// TIA Portal project "FactoryIO_Template_S7-1200_V15_V15.1" (V15.1)
// Vorlageprojekt für das Buch mit Zielsystem S7-1200

(* hardware
DEVICE "S7-1200-Station_1"  S7-1200 Station
   slot 0: "Baugruppenträger_0"  Rack  V1.0
   slot 1: "PLC_1"  CPU 1211C DC/DC/DC  6ES7 211-1AE40-0XB0  V4.1
DEVICE "HMI_1"  KTP700 Basic PN
   slot 0: "HMI_1"  KTP700 Basic PN  6AV2 123-2GB03-0AX0  15.1.0.0
   slot 1: "HMI_RT_1"  KTP700 Basic PN  6AV2 123-2GB03-0AX0  15.1.0.0
   slot 5: "HMI_1.IE_CP_1"  PROFINET Interface  15.0.1.0
      slot 1: "Interfaz PROFINET_1"  PROFINET Interface
         slot 1: "Port_1"  Port
*)

// ===== PLC "PLC_1"  CPU 1211C DC/DC/DC =====

VAR_GLOBAL   // PLC tag table "Standard-Variablentabelle"
   "Start" AT %I0.3 : Bool;
   "Reset" AT %I0.4 : Bool;
   "Stop" AT %I0.5 : Bool;
   "Auto" AT %I0.6 : Bool;
   "Emergency Stop" AT %I0.7 : Bool;
   "Buffer vel" AT %ID30 : Real;
   "At buffer entry" AT %I0.0 : Bool;
   "At buffer exit" AT %I0.1 : Bool;
   "At exit" AT %I0.2 : Bool;
   "Stop Blade" AT %Q0.0 : Bool;
   "Start Light" AT %Q0.1 : Bool;
   "Reset Light" AT %Q0.2 : Bool;
   "Stop Light" AT %Q0.3 : Bool;
   "Emitter" AT %Q0.4 : Bool;
   "Buffer Conveyor" AT %QD30 : Real;
   "Exit Conveyor" AT %QD34 : Real;
   "Counter" AT %QD38 : DInt;
   "System_Byte" AT %MB1 : Byte;
   "FirstScan" AT %M1.0 : Bool;
   "DiagStatusUpdate" AT %M1.1 : Bool;
   "AlwaysTRUE" AT %M1.2 : Bool;
   "AlwaysFALSE" AT %M1.3 : Bool;
   "System_Byte(1)" AT %MB1 : Byte;
   "Clock_Byte" AT %MB0 : Byte;
   "Clock_10Hz" AT %M0.0 : Bool;
   "Clock_5Hz" AT %M0.1 : Bool;
   "Clock_2.5Hz" AT %M0.2 : Bool;
   "Clock_2Hz" AT %M0.3 : Bool;
   "Clock_1.25Hz" AT %M0.4 : Bool;
   "Clock_1Hz" AT %M0.5 : Bool;
   "Clock_0.625Hz" AT %M0.6 : Bool;
   "Clock_0.5Hz" AT %M0.7 : Bool;
   "Started State" AT %M2.0 : Bool;
   "Reset State" AT %M2.1 : Bool;
   "Stop State" AT %M2.2 : Bool;
   "Emergency Stop State" AT %M2.3 : Bool;
   "Emergency Rearm State" AT %M2.4 : Bool;
   "Norm input" AT %MD30 : Real;
   "Half vel" AT %MD34 : Real;
   "Counter Entry" AT %MD50 : DInt;
   "Counter Exit" AT %MD54 : DInt;
   "Transitioning State" AT %M3.0 : Bool;
   "Exiting State" AT %M3.1 : Bool;
   "Forzar Entrada" AT %M2.5 : Bool;
   "Forzar Valor" AT %MD38 : Real;
   "Start HMI" AT %M2.6 : Bool;
   "Stop HMI" AT %M2.7 : Bool;
   "Tag_1" AT %M3.2 : Bool;
   "Tag_2" AT %M3.3 : Bool;
   "Tag_3" AT %MD42 : Real;
   "Tag_4" AT %MD46 : Real;
   "Tag_5" AT %MD58 : Real;
   "Tag_6" AT %MD62 : Real;
   "Tag_7" AT %MD66 : Real;
   "Tag_8" AT %MD70 : Real;
END_VAR

// folder: System blocks/Program resources

DATA_BLOCK "IEC_Timer_0_DB"   // DB1
{ S7_Optimized_Access := 'TRUE' }
AUTHOR : Simatic
FAMILY : IEC
NAME : IEC_TMR
VERSION : 1.0
// stored: InstanceOfName IEC_TIMER
"IEC_TIMER"
BEGIN
END_DATA_BLOCK

DATA_BLOCK "IEC_Counter_0_DB"   // DB2
{ S7_Optimized_Access := 'TRUE' }
AUTHOR : SIMATIC
FAMILY : IEC
NAME : DCNTR
VERSION : 1.2
// stored: InstanceOfName IEC_DCOUNTER
"IEC_DCOUNTER"
BEGIN
END_DATA_BLOCK

DATA_BLOCK "IEC_Counter_0_DB_1"   // DB3
{ S7_Optimized_Access := 'TRUE' }
AUTHOR : SIMATIC
FAMILY : IEC
NAME : DCNTR
VERSION : 1.2
// stored: InstanceOfName IEC_DCOUNTER
"IEC_DCOUNTER"
BEGIN
END_DATA_BLOCK

// folder: (top level)

FUNCTION "MHJ-PLC-Lab-Function-S71200" : Void   // FC9000, SCL
{ S7_Optimized_Access := 'TRUE' }
VERSION : 0.1
   VAR_TEMP
      rdTimeReturn : Int;
      outputTime : DTL;
      SyncVal : Byte;
      forVal : Int;
      forVal_2 : Int;
      Value : Byte;
   END_VAR
   VAR CONSTANT
      CompVal : Byte := 16#34;
      Value_01 : Byte := 16#11;
      Value_01_DW : DWord := 16#A165_D992;
      Value_02_DW : DWord := 16#58BE_4401;
   END_VAR
BEGIN

   #Value:=PEEK(area := 16#82,
        dbNumber := 0,
        byteOffset := 511);
   #Value := #Value + 1;

   POKE(area := 16#82,
        dbNumber := 0,
        byteOffset := 511,
        value := #Value);

   POKE(area:=16#81,
        dbNumber:=0,
        byteOffset:=1016,
        value:=#Value_01_DW);
   POKE(area := 16#81,
        dbNumber := 0,
        byteOffset := 1020,
        value := #Value_02_DW);

   POKE(area := 16#81,
        dbNumber := 0,
        byteOffset := 511,
        value := B#16#00);

   FOR #forVal := 0 TO 120 DO
       FOR #forVal_2:=0 TO 10 DO
           #rdTimeReturn:=RD_SYS_T(#outputTime);
           #rdTimeReturn := WR_SYS_T(#outputTime);
           #rdTimeReturn := RD_SYS_T(#outputTime);
           #rdTimeReturn := WR_SYS_T(#outputTime);
       END_FOR;
       #SyncVal:= PEEK(area := 16#81,
                      dbNumber := 0,
                      byteOffset := 511);
       IF #SyncVal = #CompVal THEN
          GOTO M_1;
       END_IF;
   END_FOR;
   RETURN;

   M_1:
   POKE(area := 16#81,
        dbNumber := 0,
        byteOffset := 511,
        value := B#16#0);
END_FUNCTION

ORGANIZATION_BLOCK "Main"   // OB1, LAD, ProgramCycle
TITLE = "Main Program Sweep (Cycle)"
{ S7_Optimized_Access := 'TRUE' }
VERSION : 0.1
   VAR_INPUT
      Initial_Call : Bool;   // Initial call of this OB
      Remanence : Bool;   // =True, if remanent data are available
   END_VAR
   VAR_TEMP   // added for the SCL form of the ladder/FBD networks
      _w1 : Bool;
      _w2 : Bool;
      _w3 : Bool;
      _w4 : Bool;
      _w5 : Bool;
      _w6 : Bool;
      _w7 : Bool;
      _w8 : Bool;
   END_VAR
BEGIN

REGION Network 1: Konnektierungsbaustein für PLC-Lab / Comunicacion con Factory IO (no tocar)
   // Im Netzwerk 1 wird der Konnektierungsbaustein für PLC-Lab aufgerufen.
   // Dieser Aufruf darf nicht entfernt werden!
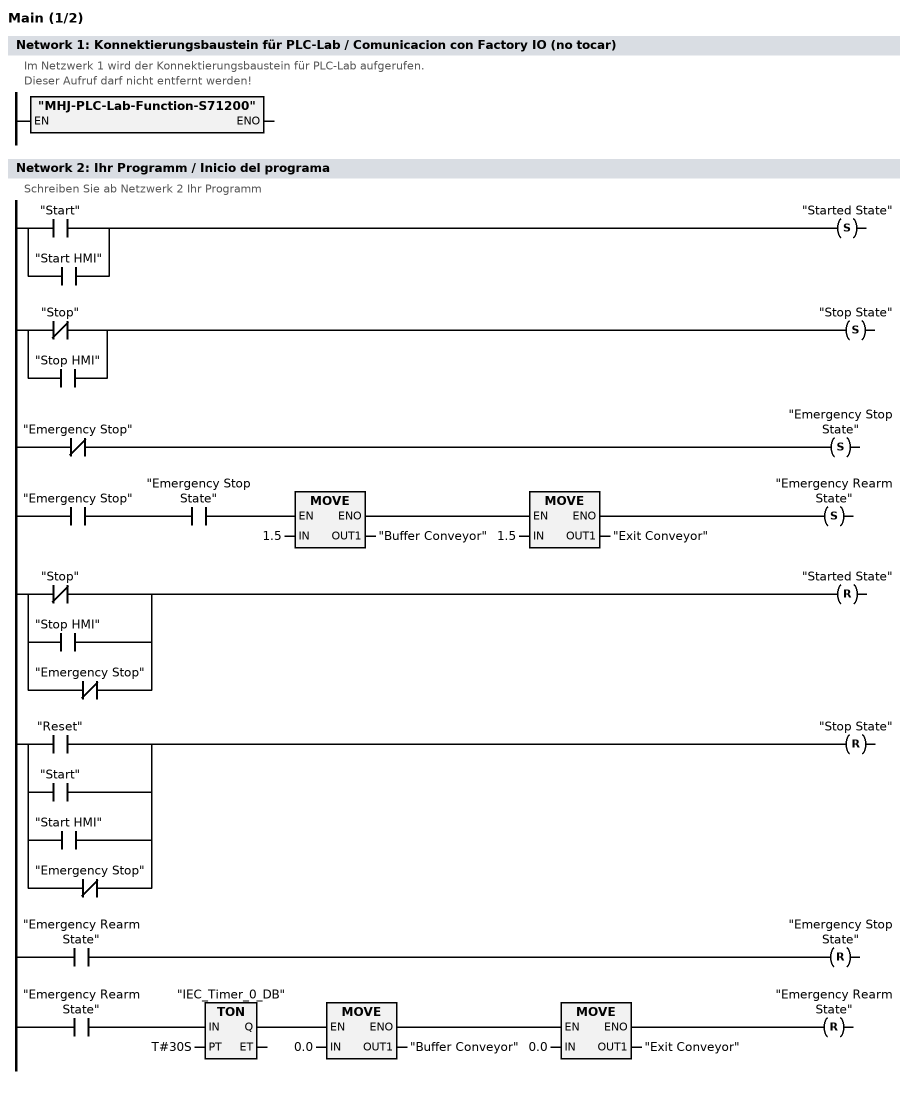
   RUNG wire#powerrail
      "MHJ-PLC-Lab-Function-S71200"()
   END_RUNG
   // the same network as SCL:
   "MHJ-PLC-Lab-Function-S71200"();
END_REGION

REGION Network 2: Ihr Programm / Inicio del programa
   // Schreiben Sie ab Netzwerk 2 Ihr Programm
   IF "Start" OR "Start HMI" THEN "Started State" := TRUE; END_IF;
   IF NOT "Stop" OR "Stop HMI" THEN "Stop State" := TRUE; END_IF;
   IF NOT "Emergency Stop" THEN "Emergency Stop State" := TRUE; END_IF;
   IF "Emergency Stop" AND "Emergency Stop State" THEN
       "Buffer Conveyor" := 1.5;
       "Exit Conveyor" := 1.5;
       "Emergency Rearm State" := TRUE;
   END_IF;
   IF NOT "Stop" OR "Stop HMI" OR NOT "Emergency Stop" THEN "Started State" := FALSE; END_IF;
   IF "Reset" OR "Start" OR "Start HMI" OR NOT "Emergency Stop" THEN "Stop State" := FALSE; END_IF;
   IF "Emergency Rearm State" THEN "Emergency Stop State" := FALSE; END_IF;
   "IEC_Timer_0_DB".TON(IN := "Emergency Rearm State", PT := T#30S);
   IF "IEC_Timer_0_DB".Q THEN
       "Buffer Conveyor" := 0.0;
       "Exit Conveyor" := 0.0;
       "Emergency Rearm State" := FALSE;
   END_IF;
END_REGION

REGION Network 3
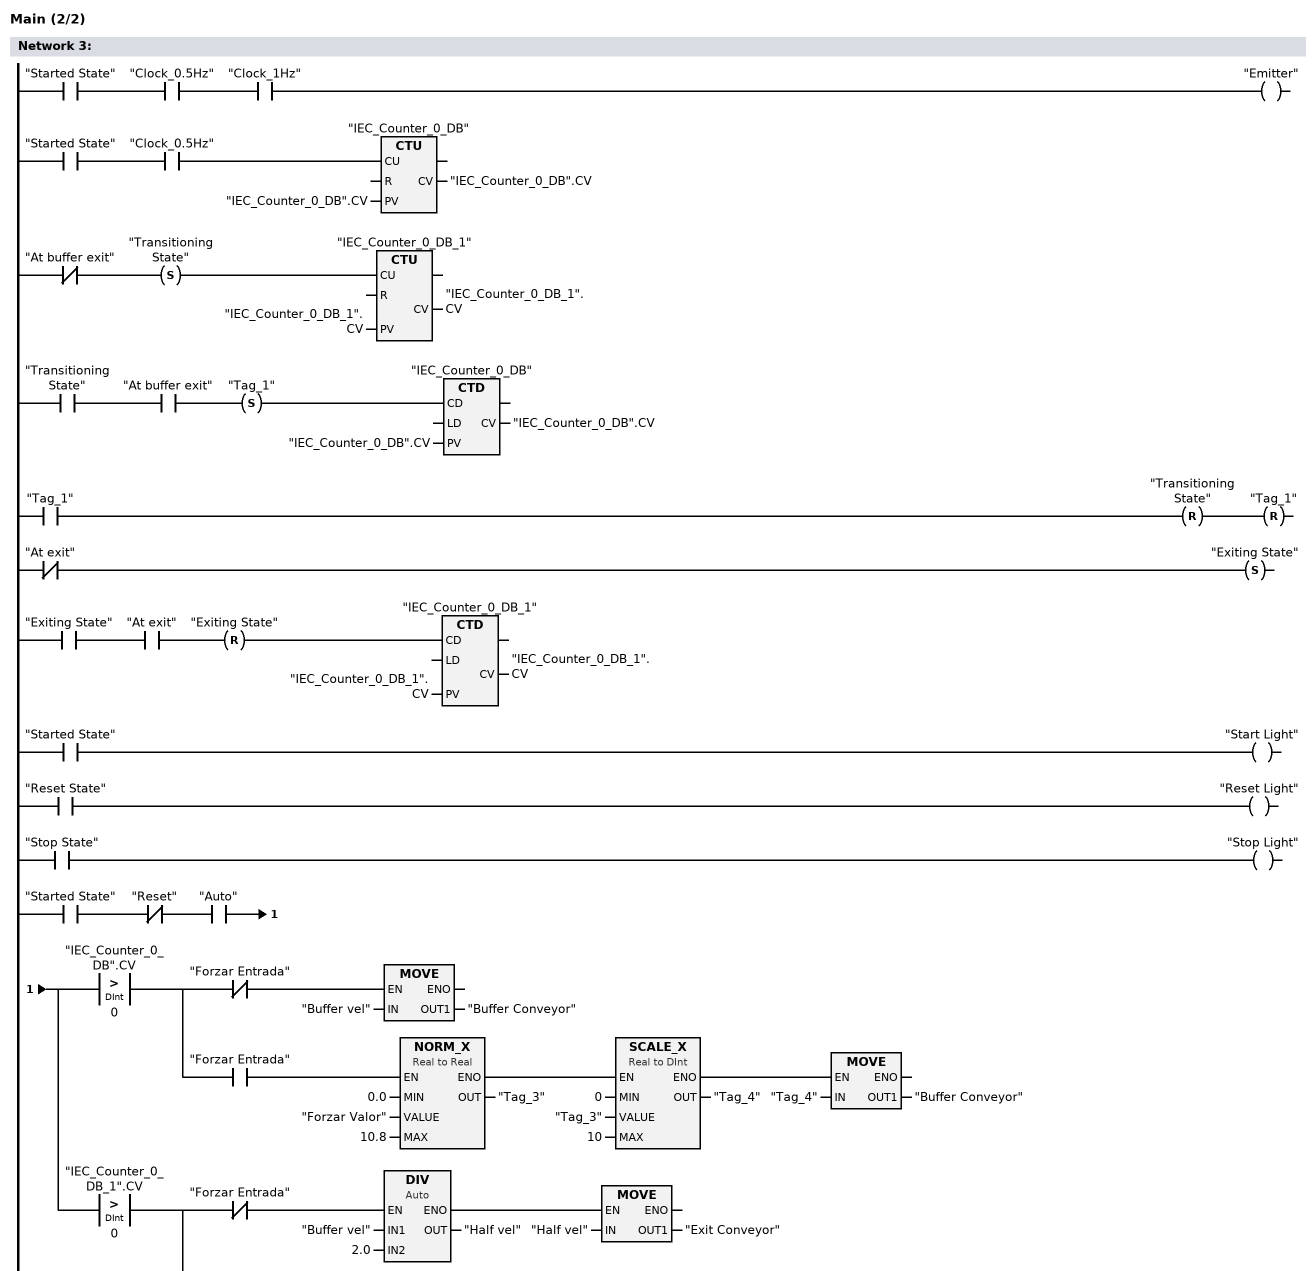
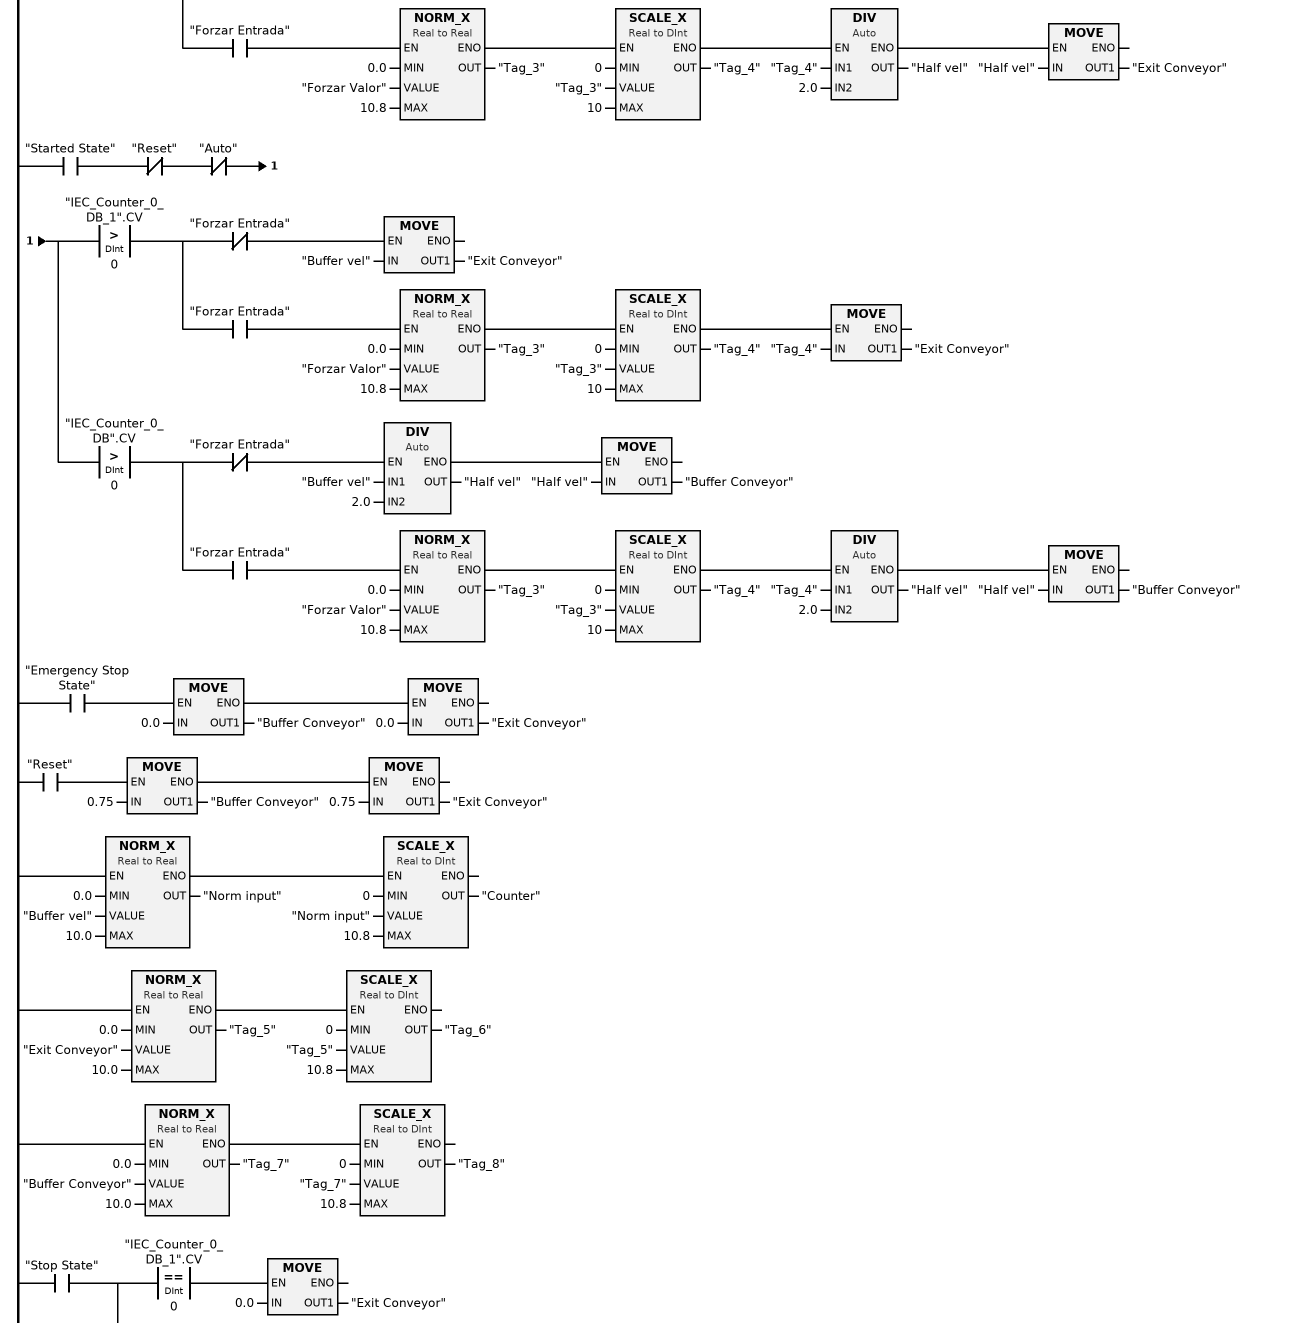
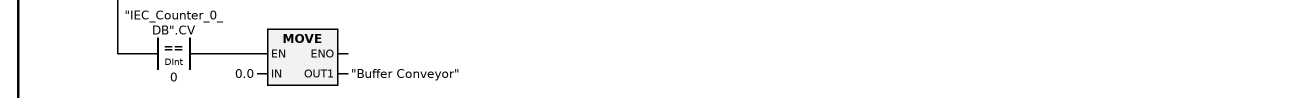
   "Emitter" := "Started State" AND "Clock_0.5Hz" AND "Clock_1Hz";
   "IEC_Counter_0_DB".CTU(CU := "Started State" AND "Clock_0.5Hz",
                          PV := "IEC_Counter_0_DB".CV,
                          CV => "IEC_Counter_0_DB".CV);
   IF NOT "At buffer exit" THEN "Transitioning State" := TRUE; END_IF;
   "IEC_Counter_0_DB_1".CTU(CU := NOT "At buffer exit",
                           PV := "IEC_Counter_0_DB_1".CV,
                           CV => "IEC_Counter_0_DB_1".CV);
   #_w1 := "Transitioning State" AND "At buffer exit";
   IF #_w1 THEN "Tag_1" := TRUE; END_IF;
   "IEC_Counter_0_DB".CTD(CD := #_w1, PV := "IEC_Counter_0_DB".CV, CV => "IEC_Counter_0_DB".CV);
   IF "Tag_1" THEN
       "Transitioning State" := FALSE;
       "Tag_1" := FALSE;
   END_IF;
   IF NOT "At exit" THEN "Exiting State" := TRUE; END_IF;
   #_w2 := "Exiting State" AND "At exit";
   IF #_w2 THEN "Exiting State" := FALSE; END_IF;
   "IEC_Counter_0_DB_1".CTD(CD := #_w2, PV := "IEC_Counter_0_DB_1".CV, CV => "IEC_Counter_0_DB_1".CV);
   "Start Light" := "Started State";
   "Reset Light" := "Reset State";
   "Stop Light" := "Stop State";
   #_w3 := "Started State" AND NOT "Reset" AND "Auto";
   #_w4 := #_w3 AND ("IEC_Counter_0_DB".CV > 0);
   IF #_w4 AND NOT "Forzar Entrada" THEN "Buffer Conveyor" := "Buffer vel"; END_IF;
   IF #_w4 AND "Forzar Entrada" THEN
       "Tag_3" := NORM_X(MIN := 0.0, VALUE := "Forzar Valor", MAX := 10.8);
       "Tag_4" := SCALE_X(MIN := 0, VALUE := "Tag_3", MAX := 10);
       "Buffer Conveyor" := "Tag_4";
   END_IF;
   #_w5 := #_w3 AND ("IEC_Counter_0_DB_1".CV > 0);
   IF #_w5 AND NOT "Forzar Entrada" THEN
       "Half vel" := "Buffer vel" / 2.0;
       "Exit Conveyor" := "Half vel";
   END_IF;
   IF #_w5 AND "Forzar Entrada" THEN
       "Tag_3" := NORM_X(MIN := 0.0, VALUE := "Forzar Valor", MAX := 10.8);
       "Tag_4" := SCALE_X(MIN := 0, VALUE := "Tag_3", MAX := 10);
       "Half vel" := "Tag_4" / 2.0;
       "Exit Conveyor" := "Half vel";
   END_IF;
   #_w6 := "Started State" AND NOT "Reset" AND NOT "Auto";
   #_w7 := #_w6 AND ("IEC_Counter_0_DB_1".CV > 0);
   IF #_w7 AND NOT "Forzar Entrada" THEN "Exit Conveyor" := "Buffer vel"; END_IF;
   IF #_w7 AND "Forzar Entrada" THEN
       "Tag_3" := NORM_X(MIN := 0.0, VALUE := "Forzar Valor", MAX := 10.8);
       "Tag_4" := SCALE_X(MIN := 0, VALUE := "Tag_3", MAX := 10);
       "Exit Conveyor" := "Tag_4";
   END_IF;
   #_w8 := #_w6 AND ("IEC_Counter_0_DB".CV > 0);
   IF #_w8 AND NOT "Forzar Entrada" THEN
       "Half vel" := "Buffer vel" / 2.0;
       "Buffer Conveyor" := "Half vel";
   END_IF;
   IF #_w8 AND "Forzar Entrada" THEN
       "Tag_3" := NORM_X(MIN := 0.0, VALUE := "Forzar Valor", MAX := 10.8);
       "Tag_4" := SCALE_X(MIN := 0, VALUE := "Tag_3", MAX := 10);
       "Half vel" := "Tag_4" / 2.0;
       "Buffer Conveyor" := "Half vel";
   END_IF;
   IF "Emergency Stop State" THEN
       "Buffer Conveyor" := 0.0;
       "Exit Conveyor" := 0.0;
   END_IF;
   IF "Reset" THEN
       "Buffer Conveyor" := 0.75;
       "Exit Conveyor" := 0.75;
   END_IF;
   "Norm input" := NORM_X(MIN := 0.0, VALUE := "Buffer vel", MAX := 10.0);
   "Counter" := SCALE_X(MIN := 0, VALUE := "Norm input", MAX := 10.8);
   "Tag_5" := NORM_X(MIN := 0.0, VALUE := "Exit Conveyor", MAX := 10.0);
   "Tag_6" := SCALE_X(MIN := 0, VALUE := "Tag_5", MAX := 10.8);
   "Tag_7" := NORM_X(MIN := 0.0, VALUE := "Buffer Conveyor", MAX := 10.0);
   "Tag_8" := SCALE_X(MIN := 0, VALUE := "Tag_7", MAX := 10.8);
   IF "Stop State" AND ("IEC_Counter_0_DB_1".CV = 0) THEN "Exit Conveyor" := 0.0; END_IF;
   IF "Stop State" AND ("IEC_Counter_0_DB".CV = 0) THEN "Buffer Conveyor" := 0.0; END_IF;
END_REGION
END_ORGANIZATION_BLOCK

(* ===== HMI "HMI_RT_1" =====
system functions are stored by id; their names below are inferred from use
connection "HMI_Conexión_1": ETHERNET, SMART_S7_1200_OMS

HMI tags "Tabla de variables estándar"
   "Exit Conveyor" : Real = PLC Tag_6 AT %MD62, 100 ms
   "Buffer Conveyor" : Real = PLC Tag_8 AT %MD70, 100 ms
   "Counter Exit" : DInt = PLC IEC_Counter_0_DB.CV AT %MD54, 100 ms
   "Counter Entry" : DInt = PLC IEC_Counter_0_DB.CV AT %MD50, 100 ms
   "Started State" : Bool = PLC "Started State" AT %M2.0, 100 ms
   "Stop State" : Bool = PLC "Stop State" AT %M2.2, 100 ms
   "Forzar Entrada" : Bool = PLC "Forzar Entrada" AT %M2.5, 100 ms
   "Forzar Valor" : Real = PLC "Forzar Valor" AT %MD38, 100 ms
   "Start HMI" : Bool = PLC "Start HMI" AT %M2.6, 100 ms
   "Stop HMI" : Bool = PLC "Stop HMI" AT %M2.7, 100 ms
   "IEC_Counter_0_DB_1_CV" : DInt = PLC IEC_Counter_0_DB_1.CV, 100 ms

Template "Plantilla_1" 800x480
   Button "Exit" at 714,429 size 71x50; TextOff 'Exit'; PictureOff "ExitRuntime_KTP700_Basic_PN_TR"; PictureOn "ExitRuntime_KTP700_Basic_PN_TR"
      on Release: StopRuntime(0)
   Button "Template_Button" at 614,429 size 71x50; TextOff 'Text'
   Button "Template_Button_1" at 514,429 size 71x50; TextOff 'Text'
   Button "Template_Button_2" at 414,429 size 71x50; TextOff 'Text'
   Button "Template_Button_3" at 314,429 size 71x50; TextOff 'Text'
   Button "Template_Button_4" at 214,429 size 71x50; TextOff 'Text'
   Button "Template_Button_5" at 114,429 size 71x50; TextOff 'Text'
   Button "Start screen" at 14,429 size 71x50; TextOff 'Start screen'; PictureOff "NavigateHome_KTP700_Basic_PN_TR"; PictureOn "NavigateHome_KTP700_Basic_PN_TR"
      on Release: ActivateScreen("Imagen raíz", 0)

screen "Imagen raíz" 800x480, template "Plantilla_1"
   Button "Botón_1" at 94,104 size 96x32; TextOff 'Start'
      on Activate: SetBit("Start HMI")
      on Deactivate: ResetBit("Start HMI")
   Circle "Círculo_1" at 120,155 size 48x48
      Appearance <- "Started State"
   Button "Botón_3" at 100,240 size 164x32; TextOff 'Forzar valor'
      on Press: SetBit("Forzar Entrada")
      on Release: ResetBit("Forzar Entrada")
   IOField "Campo ES_1" at 100,281 size 165x32; FormatPattern s999999999.999
      ProcessValue <- "Forzar Valor"
   IOField "Campo ES_2" at 405,99 size 152x32; FormatPattern s999999999.999
      ProcessValue <- "Exit Conveyor"
   TextField "Campo de texto_1" at 436,62 size 103x23; Text 'Cinta Salida'
   IOField "Campo ES_3" at 424,143 size 125x32; FormatPattern s9999999999
      ProcessValue <- "IEC_Counter_0_DB_1_CV"
   TextField "Campo de texto_2" at 370,103 size 31x23; Text 'Vel'
   TextField "Campo de texto_3" at 365,147 size 50x23; Text 'Cajas'
   IOField "Campo ES_4" at 605,99 size 165x32; FormatPattern s999999999.999
      ProcessValue <- "Buffer Conveyor"
   TextField "Campo de texto_4" at 618,62 size 117x23; Text 'Cinta Entrada'
   IOField "Campo ES_5" at 606,143 size 165x32; FormatPattern s9999999999
      ProcessValue <- "Counter Entry"
   TextField "Campo de texto_5" at 561,103 size 31x23; Text 'Vel'
   TextField "Campo de texto_6" at 549,147 size 50x23; Text 'Cajas'
   Circle "Círculo_2" at 263,155 size 48x48
      Appearance <- "Stop State"
   Button "Botón_2" at 234,104 size 96x32; TextOff 'Stop'
      on Activate: SetBit("Stop HMI")
      on Deactivate: ResetBit("Stop HMI")
*)